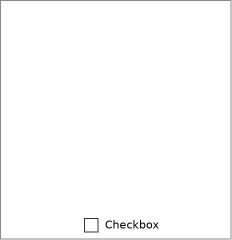
VISUALIZATION Visualization_1  // 232x240
    Checkbox (82,210 150x30), "Checkbox"
END_VISUALIZATION

(* stored: Version 1.1.0.1, ProductVersion 3.1.4024.12
   Visu Visualization_1: Id {4bf0976d-0dae-42c7-8770-a13148779d7c} *)
